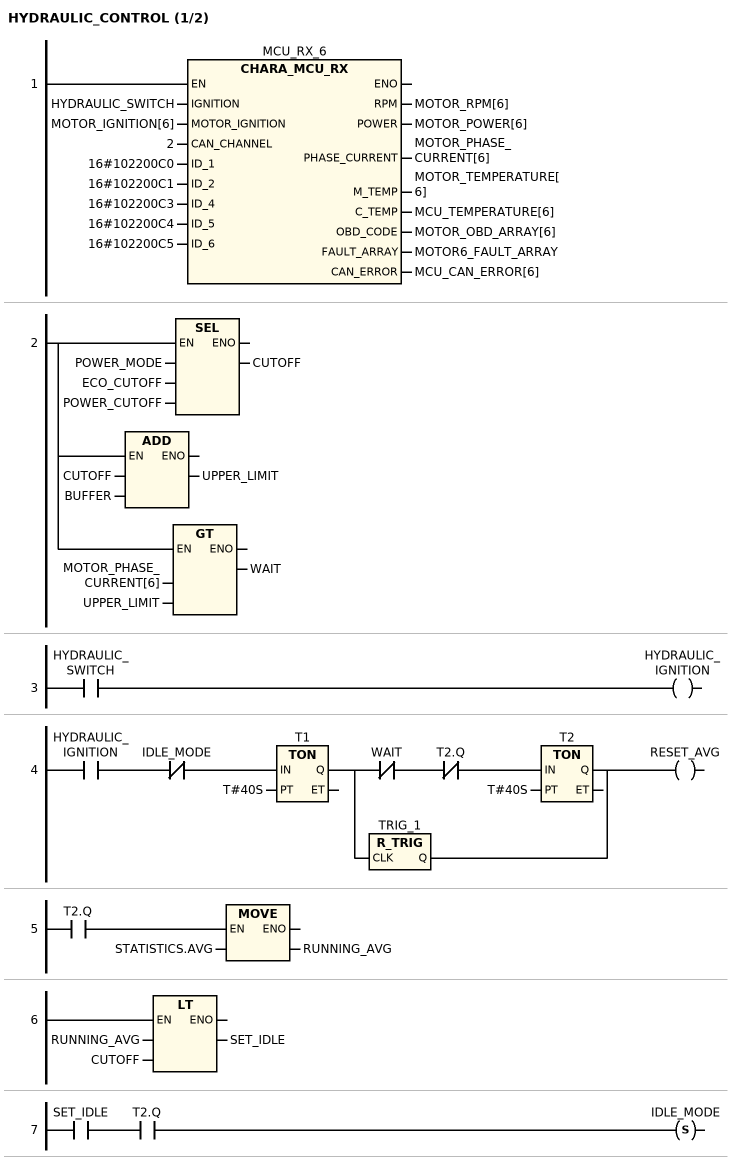
[picture p48: HYDRAULIC_CONTROL (LD)]
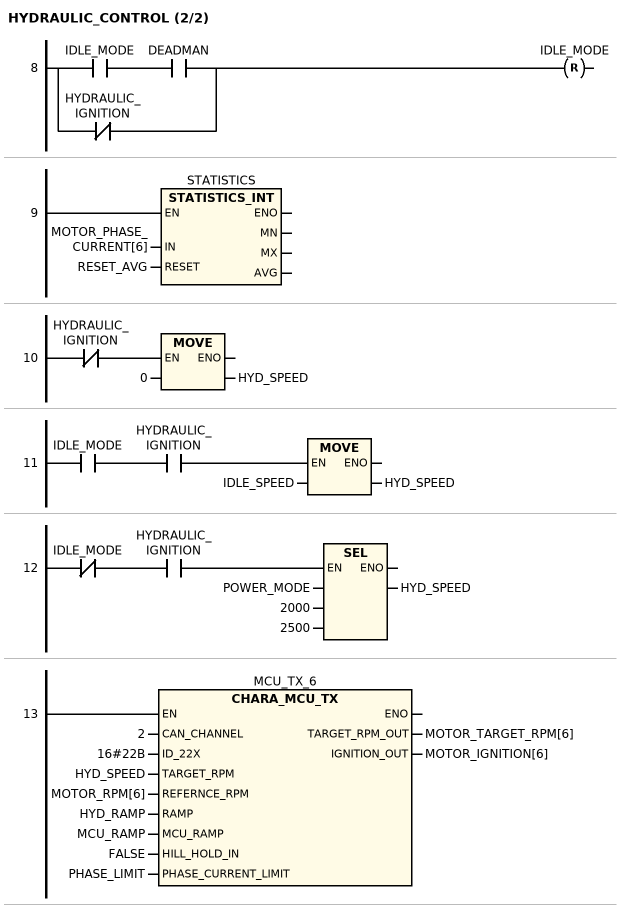
_LD_ (* Ladder Diagram *)
NETWORK 1
	*
		EN --- MCU_RX_6:CHARA_MCU_RX(IGNITION: HYDRAULIC_SWITCH, MOTOR_IGNITION: MOTOR_IGNITION[6], CAN_CHANNEL: 2, ID_1: 16#102200C0, ID_2: 16#102200C1, ID_4: 16#102200C3, ID_5: 16#102200C4, ID_6: 16#102200C5, POWER => MOTOR_POWER[6], PHASE_CURRENT => MOTOR_PHASE_CURRENT[6], M_TEMP => MOTOR_TEMPERATURE[6], C_TEMP => MCU_TEMPERATURE[6], OBD_CODE => MOTOR_OBD_ARRAY[6], FAULT_ARRAY => MOTOR6_FAULT_ARRAY, CAN_ERROR => MCU_CAN_ERROR[6]) => MOTOR_RPM[6]
NETWORK 2
	*
		EN --- SEL(POWER_MODE, ECO_CUTOFF, POWER_CUTOFF) => CUTOFF
		EN --- ADD(CUTOFF, BUFFER) => UPPER_LIMIT
		EN --- GT(MOTOR_PHASE_CURRENT[6], UPPER_LIMIT) => WAIT
NETWORK 3
	[HYDRAULIC_SWITCH] --- (HYDRAULIC_IGNITION)
NETWORK 4
	[HYDRAULIC_IGNITION] - [/IDLE_MODE] - T1:TON(IN: *, PT: T#40S) - { [/WAIT] - [/T2.Q] - T2:TON(IN: *, PT: T#40S) | TRIG_1:R_TRIG(CLK: *) } --- (RESET_AVG)
NETWORK 5
	[T2.Q]
		EN --- MOVE(STATISTICS.AVG) => RUNNING_AVG
NETWORK 6
	*
		EN --- LT(RUNNING_AVG, CUTOFF) => SET_IDLE
NETWORK 7
	[SET_IDLE] - [T2.Q] --- (S IDLE_MODE)
NETWORK 8
	{ [IDLE_MODE] - [DEADMAN] | [/HYDRAULIC_IGNITION] } --- (R IDLE_MODE)
NETWORK 9
	*
		EN --- STATISTICS:STATISTICS_INT(IN: MOTOR_PHASE_CURRENT[6], RESET: RESET_AVG)
NETWORK 10
	[/HYDRAULIC_IGNITION]
		EN --- MOVE(0) => HYD_SPEED
NETWORK 11
	[IDLE_MODE] - [HYDRAULIC_IGNITION]
		EN --- MOVE(IDLE_SPEED) => HYD_SPEED
NETWORK 12
	[/IDLE_MODE] - [HYDRAULIC_IGNITION]
		EN --- SEL(POWER_MODE, 2000, 2500) => HYD_SPEED
NETWORK 13
	*
		EN --- MCU_TX_6:CHARA_MCU_TX(CAN_CHANNEL: 2, ID_22X: 16#22B, TARGET_RPM: HYD_SPEED, REFERNCE_RPM: MOTOR_RPM[6], RAMP: HYD_RAMP, MCU_RAMP: MCU_RAMP, HILL_HOLD_IN: FALSE, PHASE_CURRENT_LIMIT: PHASE_LIMIT, IGNITION_OUT => MOTOR_IGNITION[6]) => MOTOR_TARGET_RPM[6]
_END_LD_
(* the same logic as Structured Text *)
(* Network 1 *)
MCU_RX_6(IGNITION := HYDRAULIC_SWITCH, MOTOR_IGNITION := MOTOR_IGNITION[6], CAN_CHANNEL := 2, ID_1 := 16#102200C0, ID_2 := 16#102200C1, ID_4 := 16#102200C3, ID_5 := 16#102200C4, ID_6 := 16#102200C5);
MOTOR_POWER[6] := MCU_RX_6.POWER;
MOTOR_PHASE_CURRENT[6] := MCU_RX_6.PHASE_CURRENT;
MOTOR_TEMPERATURE[6] := MCU_RX_6.M_TEMP;
MCU_TEMPERATURE[6] := MCU_RX_6.C_TEMP;
MOTOR_OBD_ARRAY[6] := MCU_RX_6.OBD_CODE;
MOTOR6_FAULT_ARRAY := MCU_RX_6.FAULT_ARRAY;
MCU_CAN_ERROR[6] := MCU_RX_6.CAN_ERROR;
MOTOR_RPM[6] := MCU_RX_6.RPM;
(* Network 2 *)
CUTOFF := SEL(POWER_MODE, ECO_CUTOFF, POWER_CUTOFF);
UPPER_LIMIT := CUTOFF + BUFFER;
WAIT := MOTOR_PHASE_CURRENT[6] > UPPER_LIMIT;
(* Network 3 *)
HYDRAULIC_IGNITION := HYDRAULIC_SWITCH;
(* Network 4 *)
T1(IN := HYDRAULIC_IGNITION AND NOT IDLE_MODE, PT := T#40S);
T2(IN := T1.Q AND NOT WAIT AND NOT T2.Q, PT := T#40S);
TRIG_1(CLK := T1.Q);
RESET_AVG := T2.Q OR TRIG_1.Q;
(* Network 5 *)
IF T2.Q THEN
	RUNNING_AVG := STATISTICS.AVG;
END_IF;
(* Network 6 *)
SET_IDLE := RUNNING_AVG < CUTOFF;
(* Network 7 *)
IF SET_IDLE AND T2.Q THEN IDLE_MODE := TRUE; END_IF;
(* Network 8 *)
IF IDLE_MODE AND DEADMAN OR NOT HYDRAULIC_IGNITION THEN IDLE_MODE := FALSE; END_IF;
(* Network 9 *)
STATISTICS(IN := MOTOR_PHASE_CURRENT[6], RESET := RESET_AVG);
(* Network 10 *)
IF NOT HYDRAULIC_IGNITION THEN
	HYD_SPEED := 0;
END_IF;
(* Network 11 *)
IF IDLE_MODE AND HYDRAULIC_IGNITION THEN
	HYD_SPEED := IDLE_SPEED;
END_IF;
(* Network 12 *)
IF NOT IDLE_MODE AND HYDRAULIC_IGNITION THEN
	HYD_SPEED := SEL(POWER_MODE, 2000, 2500);
END_IF;
(* Network 13 *)
MCU_TX_6(CAN_CHANNEL := 2, ID_22X := 16#22B, TARGET_RPM := HYD_SPEED, REFERNCE_RPM := MOTOR_RPM[6], RAMP := HYD_RAMP, MCU_RAMP := MCU_RAMP, HILL_HOLD_IN := FALSE, PHASE_CURRENT_LIMIT := PHASE_LIMIT);
MOTOR_IGNITION[6] := MCU_TX_6.IGNITION_OUT;
MOTOR_TARGET_RPM[6] := MCU_TX_6.TARGET_RPM_OUT;
END_FUNCTION_BLOCK

(* POU PROGRAM_FBs/IMU_SENSOR, LD *)
FUNCTION_BLOCK IMU_SENSOR

(*
	Created BY: Adiga
Date: 2-07-24
Version: 1
Updated BY: ADIGA
1.

*)
VAR_INPUT
END_VAR
VAR_OUTPUT
	IMY_X_OUT: BYTE;
	IMU_Y_OUT: BYTE;
	ALERT: BOOL;
END_VAR
VAR
	RX_18C: RX_CAN;
	X_ANGLE_WORD: WORD;
	X_ANGLE: INT;

	Y_ANGLE_WORD: WORD;
	Y_ANGLE: INT;

	Y_IMU: INT;
	X_IMU: INT;

	TON_IMU: TON;
	Y_ALERT: BOOL;
	PAST_TIMER: TON;
	Y_PAST: INT;
	STORE_Y_MAX: BOOL;
	X_PAST: INT;
	STORE_X_MAX: BOOL;
	STORE_Y_MIN: BOOL;
	STORE_X_MIN: BOOL;
	X_ALERT: BOOL;
	BUZZER_SOUND: BLINK;
	IMU_BUZZER: BOOL;
END_VAR
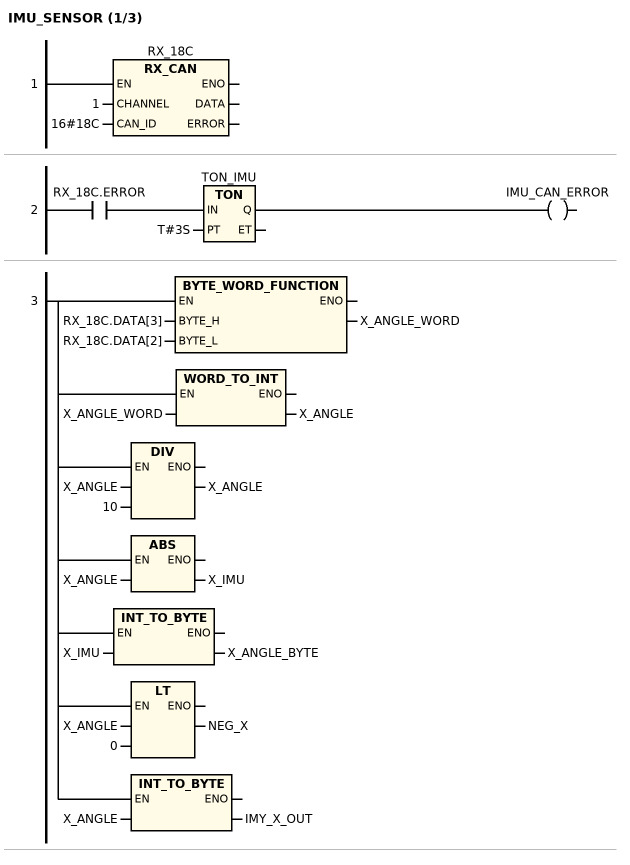
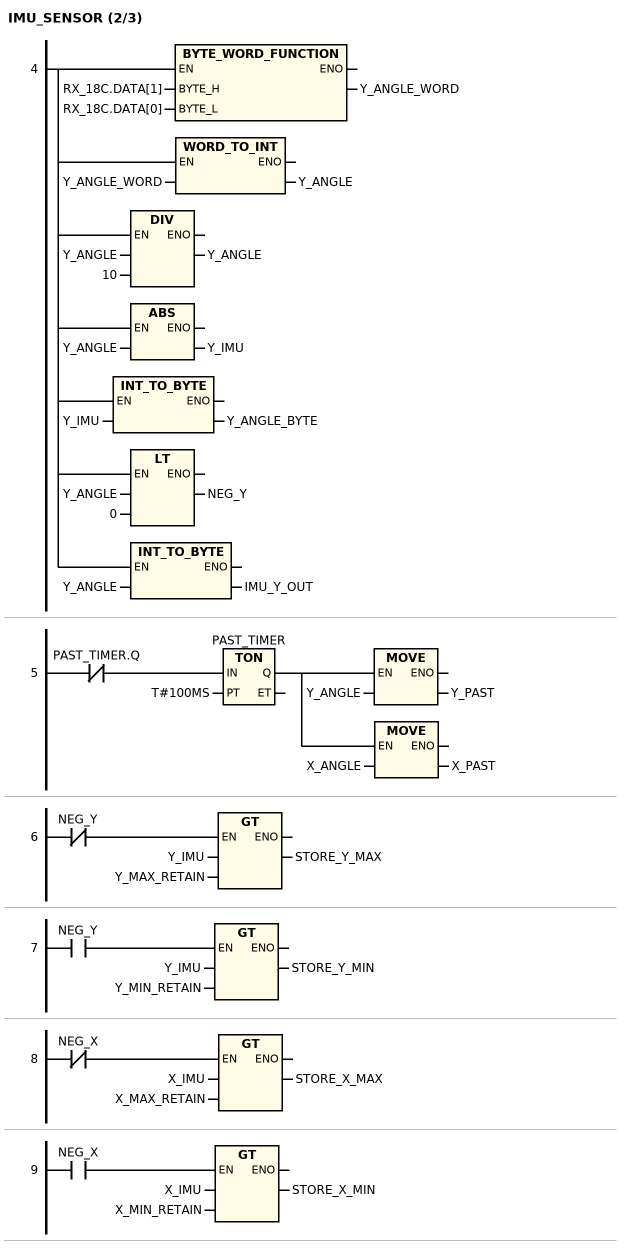
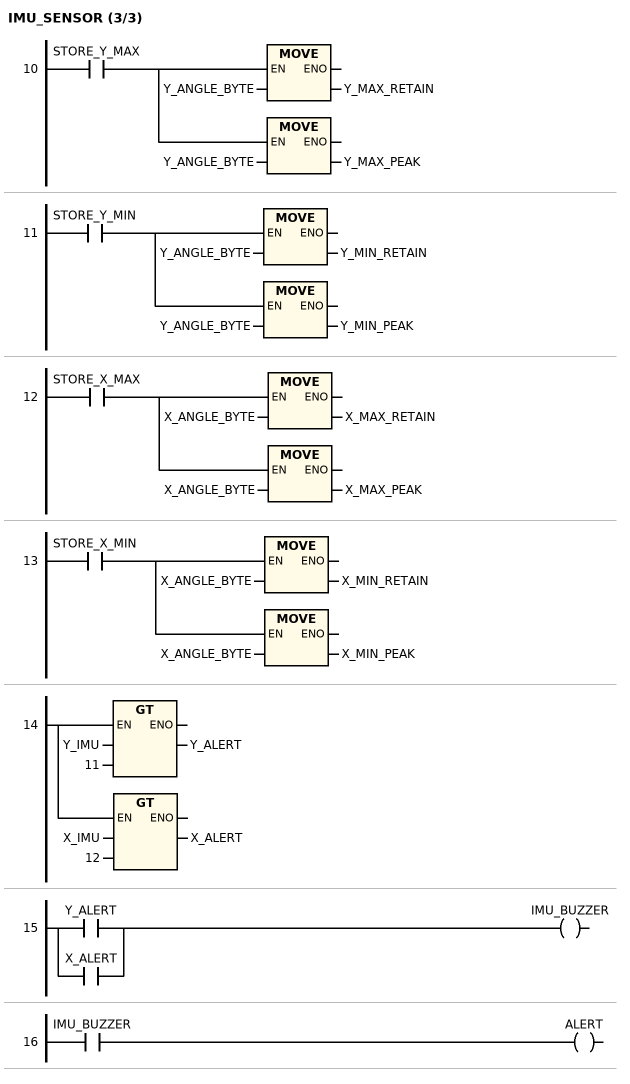
_LD_ (* Ladder Diagram *)
NETWORK 1
	*
		EN --- RX_18C:RX_CAN(CHANNEL: 1, CAN_ID: 16#18C)
NETWORK 2
	[RX_18C.ERROR] - TON_IMU:TON(IN: *, PT: T#3S) --- (IMU_CAN_ERROR)
NETWORK 3
	*
		EN --- BYTE_WORD_FUNCTION(BYTE_H: RX_18C.DATA[3], BYTE_L: RX_18C.DATA[2]) => X_ANGLE_WORD
		EN --- WORD_TO_INT(X_ANGLE_WORD) => X_ANGLE
		EN --- DIV(X_ANGLE, 10) => X_ANGLE
		EN --- ABS(X_ANGLE) => X_IMU
		EN --- INT_TO_BYTE(X_IMU) => X_ANGLE_BYTE
		EN --- LT(X_ANGLE, 0) => NEG_X
		EN --- INT_TO_BYTE(X_ANGLE) => IMY_X_OUT
NETWORK 4
	*
		EN --- BYTE_WORD_FUNCTION(BYTE_H: RX_18C.DATA[1], BYTE_L: RX_18C.DATA[0]) => Y_ANGLE_WORD
		EN --- WORD_TO_INT(Y_ANGLE_WORD) => Y_ANGLE
		EN --- DIV(Y_ANGLE, 10) => Y_ANGLE
		EN --- ABS(Y_ANGLE) => Y_IMU
		EN --- INT_TO_BYTE(Y_IMU) => Y_ANGLE_BYTE
		EN --- LT(Y_ANGLE, 0) => NEG_Y
		EN --- INT_TO_BYTE(Y_ANGLE) => IMU_Y_OUT
NETWORK 5
	[/PAST_TIMER.Q] - PAST_TIMER:TON(IN: *, PT: T#100MS)
		EN --- MOVE(Y_ANGLE) => Y_PAST
		EN --- MOVE(X_ANGLE) => X_PAST
NETWORK 6
	[/NEG_Y]
		EN --- GT(Y_IMU, Y_MAX_RETAIN) => STORE_Y_MAX
NETWORK 7
	[NEG_Y]
		EN --- GT(Y_IMU, Y_MIN_RETAIN) => STORE_Y_MIN
NETWORK 8
	[/NEG_X]
		EN --- GT(X_IMU, X_MAX_RETAIN) => STORE_X_MAX
NETWORK 9
	[NEG_X]
		EN --- GT(X_IMU, X_MIN_RETAIN) => STORE_X_MIN
NETWORK 10
	[STORE_Y_MAX]
		EN --- MOVE(Y_ANGLE_BYTE) => Y_MAX_RETAIN
		EN --- MOVE(Y_ANGLE_BYTE) => Y_MAX_PEAK
NETWORK 11
	[STORE_Y_MIN]
		EN --- MOVE(Y_ANGLE_BYTE) => Y_MIN_RETAIN
		EN --- MOVE(Y_ANGLE_BYTE) => Y_MIN_PEAK
NETWORK 12
	[STORE_X_MAX]
		EN --- MOVE(X_ANGLE_BYTE) => X_MAX_RETAIN
		EN --- MOVE(X_ANGLE_BYTE) => X_MAX_PEAK
NETWORK 13
	[STORE_X_MIN]
		EN --- MOVE(X_ANGLE_BYTE) => X_MIN_RETAIN
		EN --- MOVE(X_ANGLE_BYTE) => X_MIN_PEAK
NETWORK 14
	*
		EN --- GT(Y_IMU, 11) => Y_ALERT
		EN --- GT(X_IMU, 12) => X_ALERT
NETWORK 15
	{ [Y_ALERT] | [X_ALERT] } --- (IMU_BUZZER)
NETWORK 16
	[IMU_BUZZER] --- (ALERT)
_END_LD_
(* the same logic as Structured Text *)
(* Network 1 *)
RX_18C(CHANNEL := 1, CAN_ID := 16#18C);
(* Network 2 *)
TON_IMU(IN := RX_18C.ERROR, PT := T#3S);
IMU_CAN_ERROR := TON_IMU.Q;
(* Network 3 *)
X_ANGLE_WORD := BYTE_WORD_FUNCTION(BYTE_H := RX_18C.DATA[3], BYTE_L := RX_18C.DATA[2]);
X_ANGLE := WORD_TO_INT(X_ANGLE_WORD);
X_ANGLE := X_ANGLE / 10;
X_IMU := ABS(X_ANGLE);
X_ANGLE_BYTE := INT_TO_BYTE(X_IMU);
NEG_X := X_ANGLE < 0;
IMY_X_OUT := INT_TO_BYTE(X_ANGLE);
(* Network 4 *)
Y_ANGLE_WORD := BYTE_WORD_FUNCTION(BYTE_H := RX_18C.DATA[1], BYTE_L := RX_18C.DATA[0]);
Y_ANGLE := WORD_TO_INT(Y_ANGLE_WORD);
Y_ANGLE := Y_ANGLE / 10;
Y_IMU := ABS(Y_ANGLE);
Y_ANGLE_BYTE := INT_TO_BYTE(Y_IMU);
NEG_Y := Y_ANGLE < 0;
IMU_Y_OUT := INT_TO_BYTE(Y_ANGLE);
(* Network 5 *)
PAST_TIMER(IN := NOT PAST_TIMER.Q, PT := T#100MS);
IF PAST_TIMER.Q THEN
	Y_PAST := Y_ANGLE;
	X_PAST := X_ANGLE;
END_IF;
(* Network 6 *)
IF NOT NEG_Y THEN
	STORE_Y_MAX := Y_IMU > Y_MAX_RETAIN;
END_IF;
(* Network 7 *)
IF NEG_Y THEN
	STORE_Y_MIN := Y_IMU > Y_MIN_RETAIN;
END_IF;
(* Network 8 *)
IF NOT NEG_X THEN
	STORE_X_MAX := X_IMU > X_MAX_RETAIN;
END_IF;
(* Network 9 *)
IF NEG_X THEN
	STORE_X_MIN := X_IMU > X_MIN_RETAIN;
END_IF;
(* Network 10 *)
IF STORE_Y_MAX THEN
	Y_MAX_RETAIN := Y_ANGLE_BYTE;
	Y_MAX_PEAK := Y_ANGLE_BYTE;
END_IF;
(* Network 11 *)
IF STORE_Y_MIN THEN
	Y_MIN_RETAIN := Y_ANGLE_BYTE;
	Y_MIN_PEAK := Y_ANGLE_BYTE;
END_IF;
(* Network 12 *)
IF STORE_X_MAX THEN
	X_MAX_RETAIN := X_ANGLE_BYTE;
	X_MAX_PEAK := X_ANGLE_BYTE;
END_IF;
(* Network 13 *)
IF STORE_X_MIN THEN
	X_MIN_RETAIN := X_ANGLE_BYTE;
	X_MIN_PEAK := X_ANGLE_BYTE;
END_IF;
(* Network 14 *)
Y_ALERT := Y_IMU > 11;
X_ALERT := X_IMU > 12;
(* Network 15 *)
IMU_BUZZER := Y_ALERT OR X_ALERT;
(* Network 16 *)
ALERT := IMU_BUZZER;
END_FUNCTION_BLOCK

(* POU EXCLUDES/IMU_SENSOR_HOLD, LD *)
FUNCTION_BLOCK IMU_SENSOR_HOLD
VAR_OUTPUT
	IMY_X_OUT: BYTE;
	IMU_Y_OUT: BYTE;
	IMU_BUZZER_ALERT: BOOL;
END_VAR
VAR
	RX_18C: RX_CAN;
	X_ANGLE_WORD: WORD;
	X_ANGLE: INT;
	Y_ANGLE_WORD: WORD;
	Y_ANGLE: INT;
	Y_IMU: INT;
	X_IMU: INT;
	TON_IMU: TON;
	Y_ALERT: BOOL;
	X_ALERT: BOOL;
	PAST_TIMER: TON;
	Y_PAST: INT;
	STORE_Y_MAX: BOOL;
	X_PAST: INT;
	STORE_X_MAX: BOOL;
	STORE_Y_MIN: BOOL;
	STORE_X_MIN: BOOL;
END_VAR
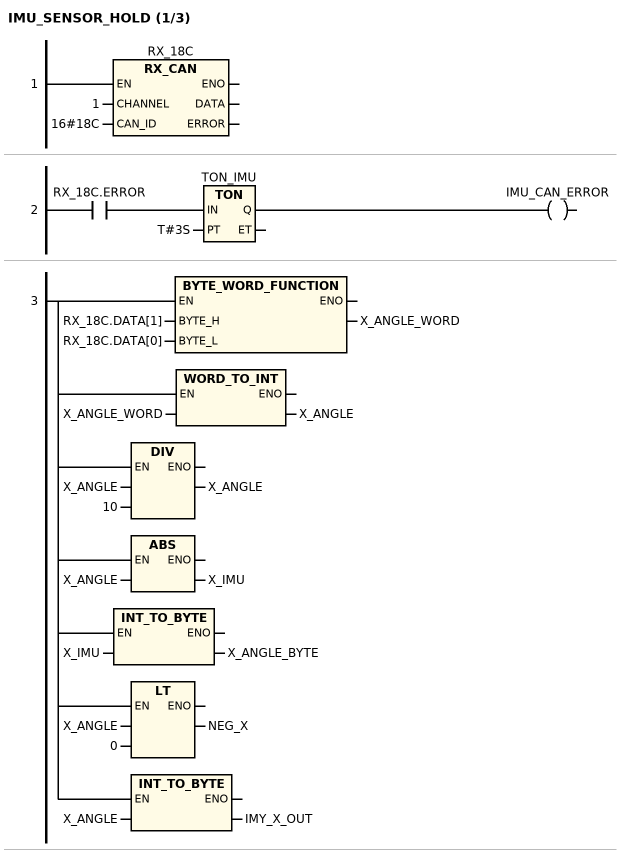
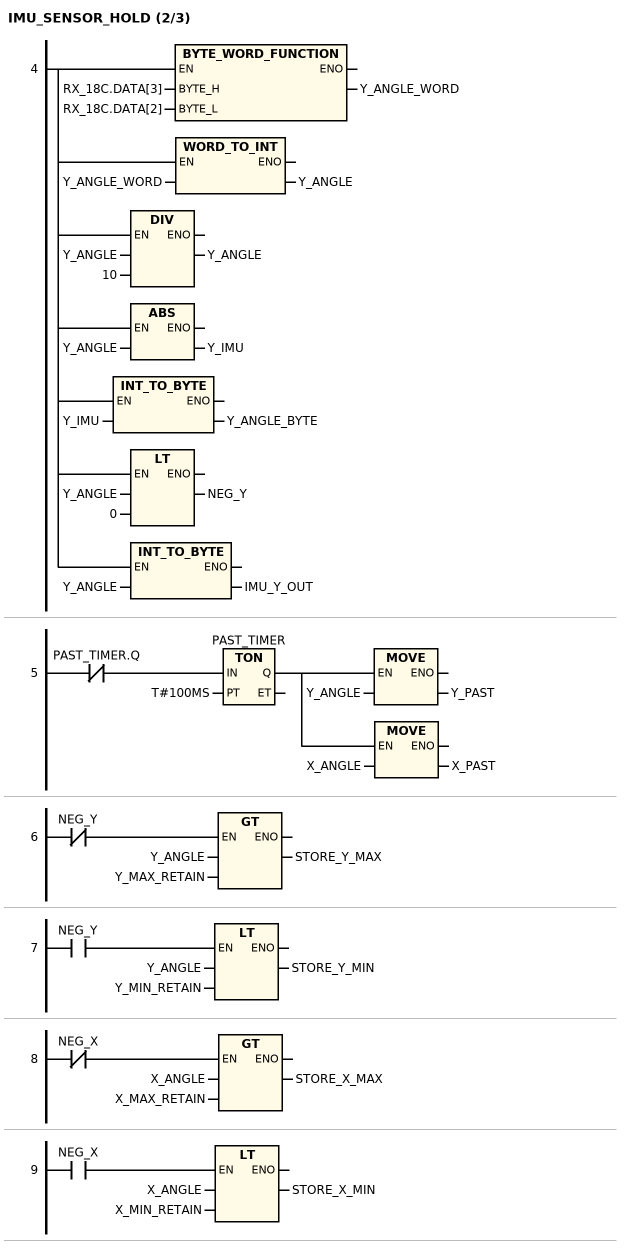
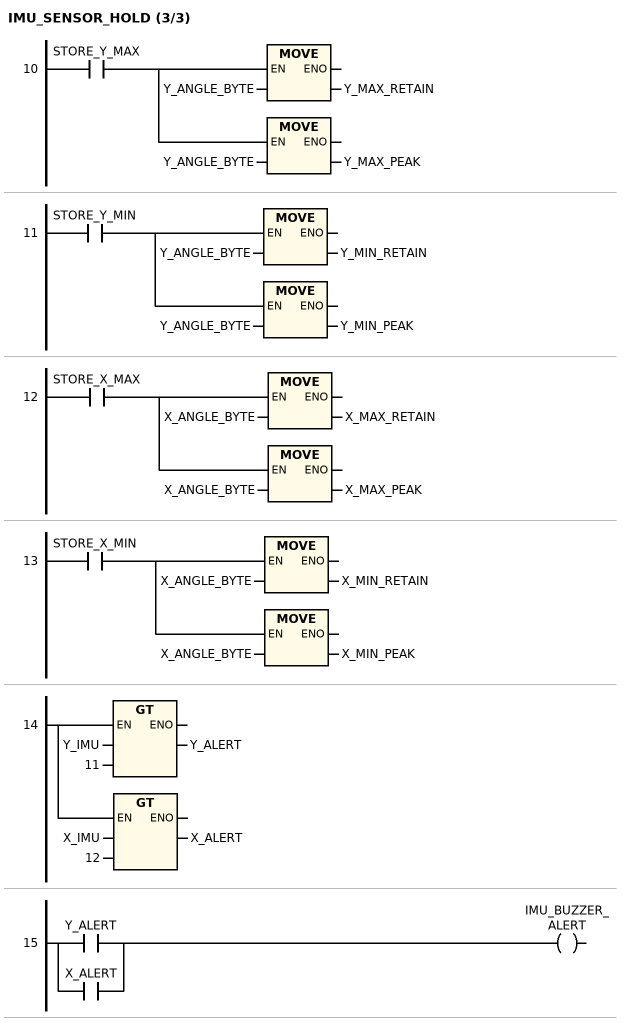
_LD_ (* Ladder Diagram *)
NETWORK 1
	*
		EN --- RX_18C:RX_CAN(CHANNEL: 1, CAN_ID: 16#18C)
NETWORK 2
	[RX_18C.ERROR] - TON_IMU:TON(IN: *, PT: T#3S) --- (IMU_CAN_ERROR)
NETWORK 3
	*
		EN --- BYTE_WORD_FUNCTION(BYTE_H: RX_18C.DATA[1], BYTE_L: RX_18C.DATA[0]) => X_ANGLE_WORD
		EN --- WORD_TO_INT(X_ANGLE_WORD) => X_ANGLE
		EN --- DIV(X_ANGLE, 10) => X_ANGLE
		EN --- ABS(X_ANGLE) => X_IMU
		EN --- INT_TO_BYTE(X_IMU) => X_ANGLE_BYTE
		EN --- LT(X_ANGLE, 0) => NEG_X
		EN --- INT_TO_BYTE(X_ANGLE) => IMY_X_OUT
NETWORK 4
	*
		EN --- BYTE_WORD_FUNCTION(BYTE_H: RX_18C.DATA[3], BYTE_L: RX_18C.DATA[2]) => Y_ANGLE_WORD
		EN --- WORD_TO_INT(Y_ANGLE_WORD) => Y_ANGLE
		EN --- DIV(Y_ANGLE, 10) => Y_ANGLE
		EN --- ABS(Y_ANGLE) => Y_IMU
		EN --- INT_TO_BYTE(Y_IMU) => Y_ANGLE_BYTE
		EN --- LT(Y_ANGLE, 0) => NEG_Y
		EN --- INT_TO_BYTE(Y_ANGLE) => IMU_Y_OUT
NETWORK 5
	[/PAST_TIMER.Q] - PAST_TIMER:TON(IN: *, PT: T#100MS)
		EN --- MOVE(Y_ANGLE) => Y_PAST
		EN --- MOVE(X_ANGLE) => X_PAST
NETWORK 6
	[/NEG_Y]
		EN --- GT(Y_ANGLE, Y_MAX_RETAIN) => STORE_Y_MAX
NETWORK 7
	[NEG_Y]
		EN --- LT(Y_ANGLE, Y_MIN_RETAIN) => STORE_Y_MIN
NETWORK 8
	[/NEG_X]
		EN --- GT(X_ANGLE, X_MAX_RETAIN) => STORE_X_MAX
NETWORK 9
	[NEG_X]
		EN --- LT(X_ANGLE, X_MIN_RETAIN) => STORE_X_MIN
NETWORK 10
	[STORE_Y_MAX]
		EN --- MOVE(Y_ANGLE_BYTE) => Y_MAX_RETAIN
		EN --- MOVE(Y_ANGLE_BYTE) => Y_MAX_PEAK
NETWORK 11
	[STORE_Y_MIN]
		EN --- MOVE(Y_ANGLE_BYTE) => Y_MIN_RETAIN
		EN --- MOVE(Y_ANGLE_BYTE) => Y_MIN_PEAK
NETWORK 12
	[STORE_X_MAX]
		EN --- MOVE(X_ANGLE_BYTE) => X_MAX_RETAIN
		EN --- MOVE(X_ANGLE_BYTE) => X_MAX_PEAK
NETWORK 13
	[STORE_X_MIN]
		EN --- MOVE(X_ANGLE_BYTE) => X_MIN_RETAIN
		EN --- MOVE(X_ANGLE_BYTE) => X_MIN_PEAK
NETWORK 14
	*
		EN --- GT(Y_IMU, 11) => Y_ALERT
		EN --- GT(X_IMU, 12) => X_ALERT
NETWORK 15
	{ [Y_ALERT] | [X_ALERT] } --- (IMU_BUZZER_ALERT)
_END_LD_
(* the same logic as Structured Text *)
(* Network 1 *)
RX_18C(CHANNEL := 1, CAN_ID := 16#18C);
(* Network 2 *)
TON_IMU(IN := RX_18C.ERROR, PT := T#3S);
IMU_CAN_ERROR := TON_IMU.Q;
(* Network 3 *)
X_ANGLE_WORD := BYTE_WORD_FUNCTION(BYTE_H := RX_18C.DATA[1], BYTE_L := RX_18C.DATA[0]);
X_ANGLE := WORD_TO_INT(X_ANGLE_WORD);
X_ANGLE := X_ANGLE / 10;
X_IMU := ABS(X_ANGLE);
X_ANGLE_BYTE := INT_TO_BYTE(X_IMU);
NEG_X := X_ANGLE < 0;
IMY_X_OUT := INT_TO_BYTE(X_ANGLE);
(* Network 4 *)
Y_ANGLE_WORD := BYTE_WORD_FUNCTION(BYTE_H := RX_18C.DATA[3], BYTE_L := RX_18C.DATA[2]);
Y_ANGLE := WORD_TO_INT(Y_ANGLE_WORD);
Y_ANGLE := Y_ANGLE / 10;
Y_IMU := ABS(Y_ANGLE);
Y_ANGLE_BYTE := INT_TO_BYTE(Y_IMU);
NEG_Y := Y_ANGLE < 0;
IMU_Y_OUT := INT_TO_BYTE(Y_ANGLE);
(* Network 5 *)
PAST_TIMER(IN := NOT PAST_TIMER.Q, PT := T#100MS);
IF PAST_TIMER.Q THEN
	Y_PAST := Y_ANGLE;
	X_PAST := X_ANGLE;
END_IF;
(* Network 6 *)
IF NOT NEG_Y THEN
	STORE_Y_MAX := Y_ANGLE > Y_MAX_RETAIN;
END_IF;
(* Network 7 *)
IF NEG_Y THEN
	STORE_Y_MIN := Y_ANGLE < Y_MIN_RETAIN;
END_IF;
(* Network 8 *)
IF NOT NEG_X THEN
	STORE_X_MAX := X_ANGLE > X_MAX_RETAIN;
END_IF;
(* Network 9 *)
IF NEG_X THEN
	STORE_X_MIN := X_ANGLE < X_MIN_RETAIN;
END_IF;
(* Network 10 *)
IF STORE_Y_MAX THEN
	Y_MAX_RETAIN := Y_ANGLE_BYTE;
	Y_MAX_PEAK := Y_ANGLE_BYTE;
END_IF;
(* Network 11 *)
IF STORE_Y_MIN THEN
	Y_MIN_RETAIN := Y_ANGLE_BYTE;
	Y_MIN_PEAK := Y_ANGLE_BYTE;
END_IF;
(* Network 12 *)
IF STORE_X_MAX THEN
	X_MAX_RETAIN := X_ANGLE_BYTE;
	X_MAX_PEAK := X_ANGLE_BYTE;
END_IF;
(* Network 13 *)
IF STORE_X_MIN THEN
	X_MIN_RETAIN := X_ANGLE_BYTE;
	X_MIN_PEAK := X_ANGLE_BYTE;
END_IF;
(* Network 14 *)
Y_ALERT := Y_IMU > 11;
X_ALERT := X_IMU > 12;
(* Network 15 *)
IMU_BUZZER_ALERT := Y_ALERT OR X_ALERT;
END_FUNCTION_BLOCK

(* POU PROGRAM_FBs/MAKERSAN_JOYSTICK, LD *)
FUNCTION_BLOCK MAKERSAN_JOYSTICK
(*
Created by: SR Karthik Raju
Date: 23-09-24
Version: 1
Updated by:
Update date:
Description: This block reads the Makersan joystick data from the CAN.
*)
VAR_INPUT
	CAN_CHANNEL: BYTE;
END_VAR
VAR_OUTPUT
	JX: INT;
	JY: INT;
	LEFT_BUTTON: BOOL;
	RIGHT_BUTTON: BOOL;
	DEADMAN: BOOL;
	AXIS_POSITION: ARRAY [0..4] OF BOOL;
	CAN_ERROR: BOOL;
END_VAR
VAR
	RX_284: RX_CAN;
	RX_184: RX_CAN;
	TON_1: TON;
	X_WORD: WORD;
	Y_WORD: WORD;
	JX_INT: INT;
	JY_INT: INT;
	JY_ORIGIN: BOOL;
	JX_ORIGIN: BOOL;
END_VAR
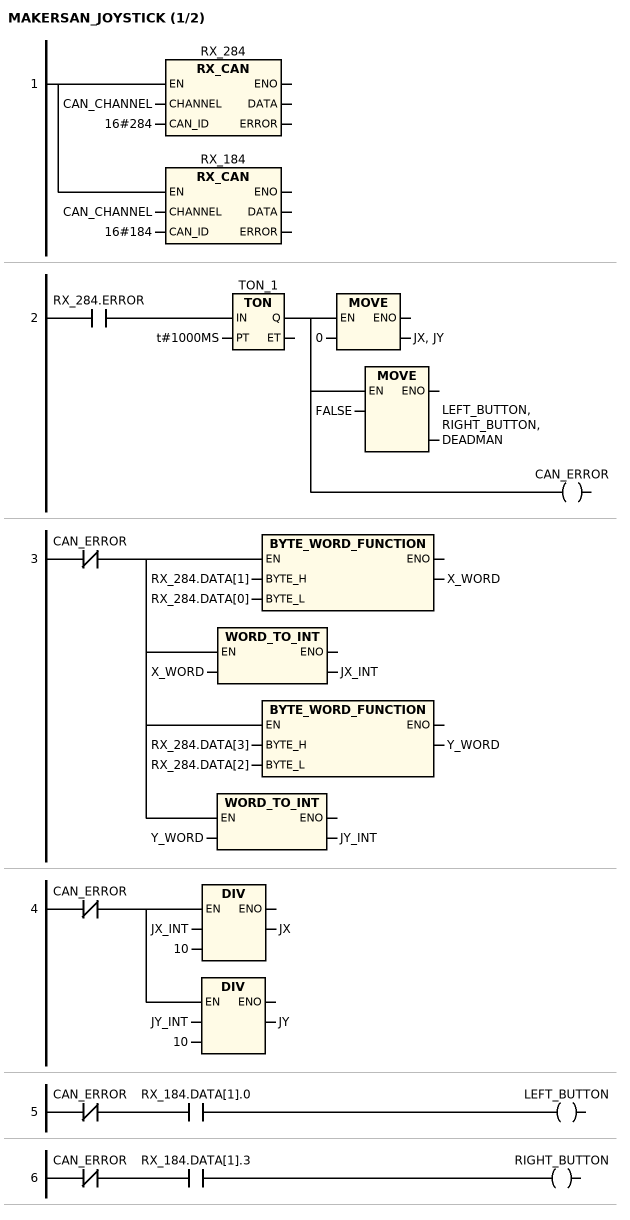
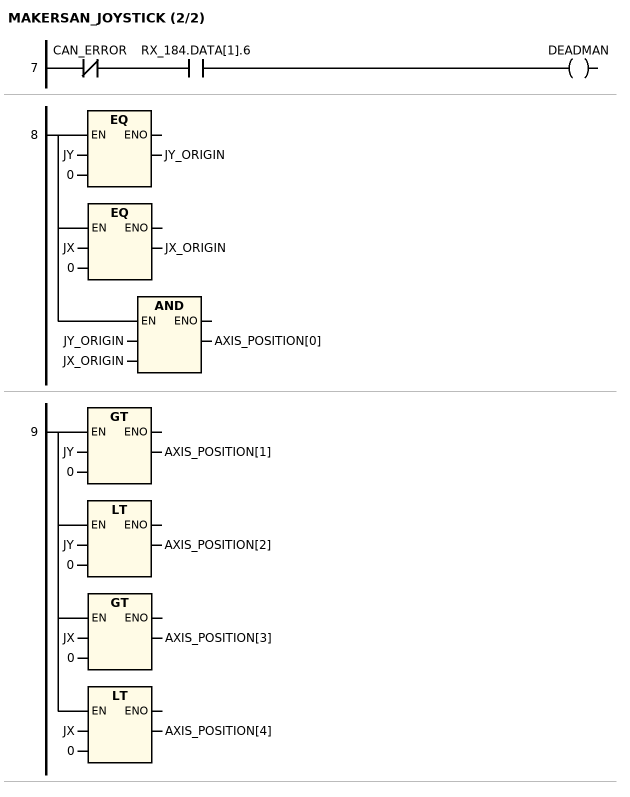
_LD_ (* Ladder Diagram *)
NETWORK 1
	*
		EN --- RX_284:RX_CAN(CHANNEL: CAN_CHANNEL, CAN_ID: 16#284)
		EN --- RX_184:RX_CAN(CHANNEL: CAN_CHANNEL, CAN_ID: 16#184)
NETWORK 2
	[RX_284.ERROR] - TON_1:TON(IN: *, PT: t#1000MS) --- (CAN_ERROR)
		EN --- MOVE(0) => JX, JY
		EN --- MOVE(FALSE) => LEFT_BUTTON, RIGHT_BUTTON, DEADMAN
NETWORK 3
	[/CAN_ERROR]
		EN --- BYTE_WORD_FUNCTION(BYTE_H: RX_284.DATA[1], BYTE_L: RX_284.DATA[0]) => X_WORD
		EN --- WORD_TO_INT(X_WORD) => JX_INT
		EN --- BYTE_WORD_FUNCTION(BYTE_H: RX_284.DATA[3], BYTE_L: RX_284.DATA[2]) => Y_WORD
		EN --- WORD_TO_INT(Y_WORD) => JY_INT
NETWORK 4
	[/CAN_ERROR]
		EN --- DIV(JX_INT, 10) => JX
		EN --- DIV(JY_INT, 10) => JY
NETWORK 5
	[/CAN_ERROR] - [RX_184.DATA[1].0] --- (LEFT_BUTTON)
NETWORK 6
	[/CAN_ERROR] - [RX_184.DATA[1].3] --- (RIGHT_BUTTON)
NETWORK 7
	[/CAN_ERROR] - [RX_184.DATA[1].6] --- (DEADMAN)
NETWORK 8
	*
		EN --- EQ(JY, 0) => JY_ORIGIN
		EN --- EQ(JX, 0) => JX_ORIGIN
		EN --- AND(JY_ORIGIN, JX_ORIGIN) => AXIS_POSITION[0]
NETWORK 9
	*
		EN --- GT(JY, 0) => AXIS_POSITION[1]
		EN --- LT(JY, 0) => AXIS_POSITION[2]
		EN --- GT(JX, 0) => AXIS_POSITION[3]
		EN --- LT(JX, 0) => AXIS_POSITION[4]
_END_LD_
(* the same logic as Structured Text *)
(* Network 1 *)
RX_284(CHANNEL := CAN_CHANNEL, CAN_ID := 16#284);
RX_184(CHANNEL := CAN_CHANNEL, CAN_ID := 16#184);
(* Network 2: see the listing above *)
(* Network 3 *)
IF NOT CAN_ERROR THEN
	X_WORD := BYTE_WORD_FUNCTION(BYTE_H := RX_284.DATA[1], BYTE_L := RX_284.DATA[0]);
	JX_INT := WORD_TO_INT(X_WORD);
	Y_WORD := BYTE_WORD_FUNCTION(BYTE_H := RX_284.DATA[3], BYTE_L := RX_284.DATA[2]);
	JY_INT := WORD_TO_INT(Y_WORD);
END_IF;
(* Network 4 *)
IF NOT CAN_ERROR THEN
	JX := JX_INT / 10;
	JY := JY_INT / 10;
END_IF;
(* Network 5 *)
LEFT_BUTTON := NOT CAN_ERROR AND RX_184.DATA[1].0;
(* Network 6 *)
RIGHT_BUTTON := NOT CAN_ERROR AND RX_184.DATA[1].3;
(* Network 7 *)
DEADMAN := NOT CAN_ERROR AND RX_184.DATA[1].6;
(* Network 8 *)
JY_ORIGIN := JY = 0;
JX_ORIGIN := JX = 0;
AXIS_POSITION[0] := JY_ORIGIN AND JX_ORIGIN;
(* Network 9 *)
AXIS_POSITION[1] := JY > 0;
AXIS_POSITION[2] := JY < 0;
AXIS_POSITION[3] := JX > 0;
AXIS_POSITION[4] := JX < 0;
END_FUNCTION_BLOCK

(* POU FUNCTIONS/MAP_INT, ST *)
FUNCTION MAP_INT : INT
(*
Created By: Nikshitha S
Date: 10-08-2023
Version: 1
Description: This function block maps the Input value range to the Output value range for the values in INT datatype.
Thus, consuming less memory than the library block "LIN_TRAFO" which uses REAL datatype.
*)
VAR_INPUT
	IN: INT;
	IN_MIN:INT;
	IN_MAX : INT;
	OUT_MIN:INT;
	OUT_MAX:INT;
END_VAR
VAR
	ERROR: BOOL;
	FINAL_MAP: INT;
	INPUT_RANGE: INT;
	OUTPUT_RANGE: INT;
END_VAR
ERROR := (IN_MAX-IN_MIN=0) OR (IN<IN_MIN) OR (IN>IN_MAX);
INPUT_RANGE := IN_MAX-IN_MIN;
OUTPUT_RANGE := OUT_MAX-OUT_MIN;
MAP_INT:= ((IN-IN_MIN)*OUTPUT_RANGE) / INPUT_RANGE + OUT_MIN;
IF ERROR AND (IN<IN_MIN)THEN
MAP_INT:=OUT_MIN;
END_IF
IF ERROR AND (IN>IN_MAX)THEN
MAP_INT:=OUT_MAX;
END_IF
END_FUNCTION

(* POU EXCLUDES/MAP_REAL, ST *)
FUNCTION MAP_REAL : REAL
(*
Created By: Bhagyesh
Date: Nov - 2021
Description: This function block maps the Input value range to the Output value range for the values in REAL datatype.
*)
VAR_INPUT
	IN: REAL;				(* input value*)
	IN_MIN:REAL;			(* minimum input value *)
	IN_MAX:REAL;			(* maximum input value *)
	OUT_MIN:REAL;		(* corresponding minimum output value *)
	OUT_MAX:REAL;		(* corresponding maximum output value *)
END_VAR
VAR
	Diff: REAL;
	ERROR: BOOL;		(* error: IN_MIN = IN_MAX or IN out of interval *)
END_VAR
Diff := IN_MAX-IN_MIN;
ERROR := (Diff=0) OR (IN<IN_MIN) OR (IN>IN_MAX);
MAP_REAL:= (IN-IN_MIN)/Diff * (OUT_MAX-OUT_MIN) + OUT_MIN;
IF ERROR AND (IN<IN_MIN)THEN
MAP_REAL:=OUT_MIN;
END_IF
IF ERROR AND (IN>IN_MAX)THEN
MAP_REAL:=OUT_MAX;
END_IF
END_FUNCTION

(* POU PROGRAM_FBs/THROTTLE_LOGIC, LD *)
FUNCTION_BLOCK THROTTLE_LOGIC
(*
Author: Bhagyesh
Description: This function block takes the joystick input from the RunLogic block and calculates the throttle for each side of the motors based on the turning logic.
This function block also implements the Zero degree turn.
*)
VAR_INPUT
	JX_IN: INT;
	JY_IN: INT;
	MCUBRAKE: BOOL;
	RPM_FACTOR_IN: INT;
END_VAR
VAR_OUTPUT
	THR_L: INT;
	THR_R: INT;
END_VAR
VAR
	THR_1: INT;
	THR_2: INT;
	THR_R_INTER: INT;
	SET_FWD: BOOL;
	SET_REV: BOOL;
	SET_RIGHT_ZERO: BOOL;
	SET_LEFT_ZERO: BOOL;

	JOY_ORIGIN: BOOL;
	FWD: BOOL;
	REV: BOOL;
	RIGHT_ZERO: BOOL;
	LEFT_ZERO: BOOL;
END_VAR
VAR CONSTANT

END_VAR
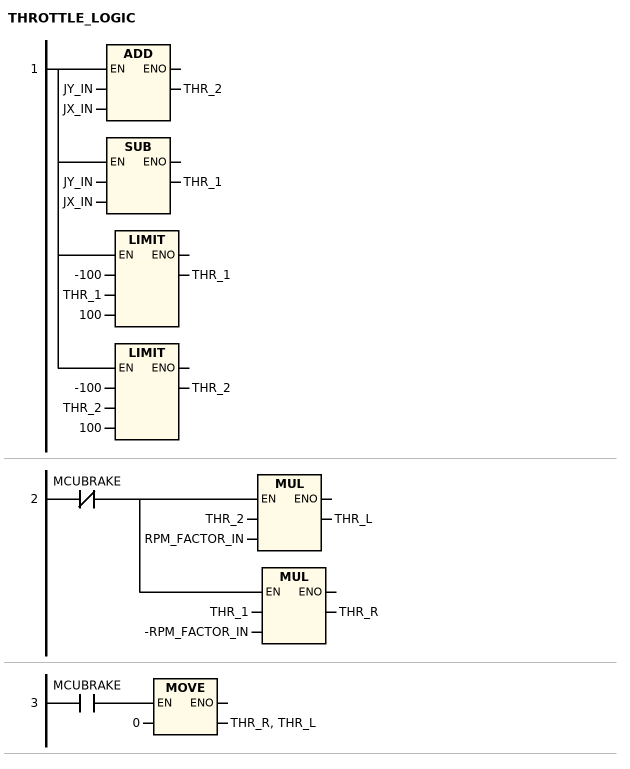
_LD_ (* Ladder Diagram *)
NETWORK 1
	*
		EN --- ADD(JY_IN, JX_IN) => THR_2
		EN --- SUB(JY_IN, JX_IN) => THR_1
		EN --- LIMIT(-100, THR_1, 100) => THR_1
		EN --- LIMIT(-100, THR_2, 100) => THR_2
NETWORK 2
	[/MCUBRAKE]
		EN --- MUL(THR_2, RPM_FACTOR_IN) => THR_L
		EN --- MUL(THR_1, -RPM_FACTOR_IN) => THR_R
NETWORK 3
	[MCUBRAKE]
		EN --- MOVE(0) => THR_R, THR_L
_END_LD_
(* the same logic as Structured Text *)
(* Network 1 *)
THR_2 := JY_IN + JX_IN;
THR_1 := JY_IN - JX_IN;
THR_1 := LIMIT(-100, THR_1, 100);
THR_2 := LIMIT(-100, THR_2, 100);
(* Network 2 *)
IF NOT MCUBRAKE THEN
	THR_L := THR_2 * RPM_FACTOR_IN;
	THR_R := THR_1 * (-RPM_FACTOR_IN);
END_IF;
(* Network 3: see the listing above *)
END_FUNCTION_BLOCK

(* Visualisation GLX_v3
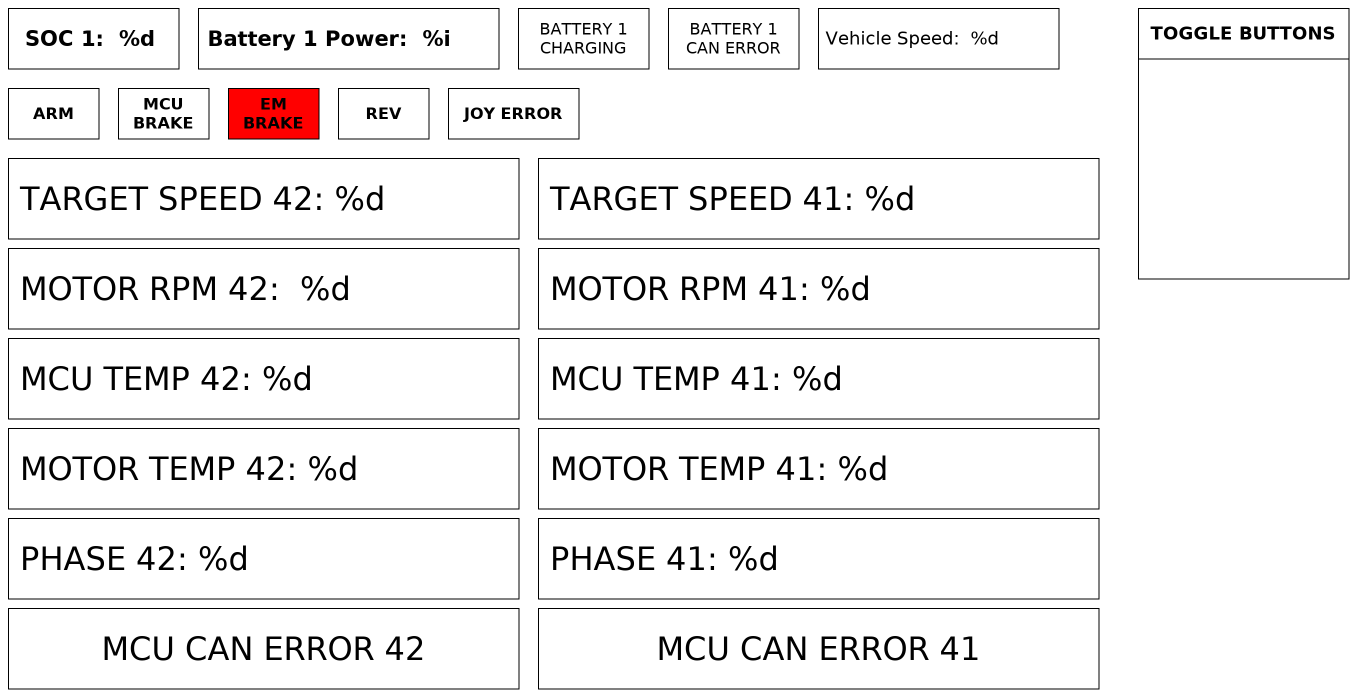
rounded rectangle at (10,10)-(181,71): text "SOC 1:  %d"; shows .BATTERY1_SOC
rounded rectangle at (200,10)-(501,71): text "Battery 1 Power:  %i"; shows .BATTERY1_POWER
rounded rectangle at (820,10)-(1061,71): text "Vehicle Speed:  %d"; shows .SPEED
rounded rectangle at (10,90)-(101,141): text "ARM"; alarm colour if .MCU_IGNITION
rounded rectangle at (120,90)-(211,141): text "MCU / BRAKE"; alarm colour if .MCU_BRAKE
rounded rectangle at (230,90)-(321,141): text "EM / BRAKE"; alarm colour if .EM_BRAKE
rounded rectangle at (540,250)-(1101,331): text "MOTOR RPM 41: %d"; shows .MOTOR_RPM[1]
rounded rectangle at (10,250)-(521,331): text "MOTOR RPM 42:  %d"; shows .MOTOR_RPM[2]
rounded rectangle at (540,340)-(1101,421): text "MCU TEMP 41: %d"; shows .MCU_TEMPERATURE[1]
rounded rectangle at (10,340)-(521,421): text "MCU TEMP 42: %d"; shows .MCU_TEMPERATURE[2]
rounded rectangle at (540,520)-(1101,601): text "PHASE 41: %d"; shows .MOTOR_PHASE_CURRENT[1]
rounded rectangle at (10,520)-(521,601): text "PHASE 42: %d"; shows .MOTOR_PHASE_CURRENT[2]
rounded rectangle at (540,160)-(1101,241): text "TARGET SPEED 41: %d"; shows .MOTOR_TARGET_RPM[1]
rounded rectangle at (10,160)-(521,241): text "TARGET SPEED 42: %d"; shows .MOTOR_TARGET_RPM[2]
rounded rectangle at (450,90)-(581,141): text "JOY ERROR"; alarm colour if .JOY_ERROR
rounded rectangle at (10,610)-(521,691): text "MCU CAN ERROR 42"; alarm colour if .MCU_CAN_ERROR[2]
rounded rectangle at (670,10)-(801,71): text "BATTERY 1 / CAN ERROR"; alarm colour if .BATTERY1_CAN_ERROR
rounded rectangle at (340,90)-(431,141): text "REV"; alarm colour if .REVERSE
rounded rectangle at (520,10)-(651,71): text "BATTERY 1 / CHARGING"; alarm colour if .BATTERY1_CHARGING
rounded rectangle at (540,610)-(1101,691): text "MCU CAN ERROR 41"; alarm colour if .MCU_CAN_ERROR[1]
rounded rectangle at (540,430)-(1101,511): text "MOTOR TEMP 41: %d"; shows .MOTOR_TEMPERATURE[1]
rounded rectangle at (10,430)-(521,511): text "MOTOR TEMP 42: %d"; shows .MOTOR_TEMPERATURE[2]
rectangle at (1140,10)-(1351,61): text "TOGGLE BUTTONS"
1 more shapes without text or variables
*)
